KUKA KRL program: chk_w2_grp4_clo.src, chk_w2_grp4_clo.dat

--- chk_w2_grp4_clo.src ---
&ACCESS RV2
&REL 12
&COMMENT Check grampos Z4 fechado
&PARAM DISKPATH = Program/SubeRotine
&PARAM TEMPLATE = C:\KRC\Roboter\Template\vorgabe
&PARAM EDITMASK = *
DEF chk_w2_grp4_clo( )
;FOLD ; Programa de verificacao de grampos Z4 fechado;%{PE}%R 4.1.16,%MKUKATPBASIS,%CCOMMENT,%VNORMAL,%P 2:Programa de verificacao de grampos Z4 fechado
;ENDFOLD

$TIMER[10] = 0
$TIMER_STOP[10] = FALSE

;FOLD WAIT FOR ( NOT IN 497 'Pres pc 1 Axor_Atego/ ACTROS Z4.1 OPN' );%{PE}%R 8.2.24,%MKUKATPBASIS,%CEXT_WAIT_FOR,%VEXT_WAIT_FOR,%P 2:, 4:NOT, 5:$IN, 6:497, 7:Pres pc 1 Axor_Atego/ ACTROS Z4.1 OPN, 9:
WAIT FOR  (  NOT $IN[497] )
;ENDFOLD
;FOLD WAIT FOR ( NOT IN 511 'ACTROS Z4.2 OPN' );%{PE}%R 8.2.24,%MKUKATPBASIS,%CEXT_WAIT_FOR,%VEXT_WAIT_FOR,%P 2:, 4:NOT, 5:$IN, 6:511, 7:ACTROS Z4.2 OPN, 9:
WAIT FOR  (  NOT $IN[511] )
;ENDFOLD
;FOLD WAIT FOR ( NOT IN 517 'Z4.2 ABERTO/ ACTROS Z4.3 OPN' );%{PE}%R 8.2.24,%MKUKATPBASIS,%CEXT_WAIT_FOR,%VEXT_WAIT_FOR,%P 2:, 4:NOT, 5:$IN, 6:517, 7:Z4.2 ABERTO/ ACTROS Z4.3 OPN, 9:
WAIT FOR  (  NOT $IN[517] )
;ENDFOLD
;FOLD WAIT FOR ( NOT IN 519 'Z4.3 ABERTO/ ACTROS Z4.4 OPN' );%{PE}%R 8.2.24,%MKUKATPBASIS,%CEXT_WAIT_FOR,%VEXT_WAIT_FOR,%P 2:, 4:NOT, 5:$IN, 6:519, 7:Z4.3 ABERTO/ ACTROS Z4.4 OPN, 9:
WAIT FOR  (  NOT $IN[519] )
;ENDFOLD
;FOLD WAIT FOR ( IN 498 'Pres pc 2 Axor_Atego/ ACTROS Z4.1 CLO' );%{PE}%R 8.2.24,%MKUKATPBASIS,%CEXT_WAIT_FOR,%VEXT_WAIT_FOR,%P 2:, 4:, 5:$IN, 6:498, 7:Pres pc 2 Axor_Atego/ ACTROS Z4.1 CLO, 9:
WAIT FOR  ( $IN[498] )
;ENDFOLD
;FOLD WAIT FOR ( IN 512 'ACTROS Z4.2 CLO' );%{PE}%R 8.2.24,%MKUKATPBASIS,%CEXT_WAIT_FOR,%VEXT_WAIT_FOR,%P 2:, 4:, 5:$IN, 6:512, 7:ACTROS Z4.2 CLO, 9:
WAIT FOR  ( $IN[512] )
;ENDFOLD
;FOLD WAIT FOR ( IN 518 'Z4.2 FECHADO/ ACTROS Z4.3 CLO' );%{PE}%R 8.2.24,%MKUKATPBASIS,%CEXT_WAIT_FOR,%VEXT_WAIT_FOR,%P 2:, 4:, 5:$IN, 6:518, 7:Z4.2 FECHADO/ ACTROS Z4.3 CLO, 9:
WAIT FOR  ( $IN[518] )
;ENDFOLD
;FOLD WAIT FOR ( IN 520 'Z4.3 FECHADO/ ACTROS Z4.4 CLO' );%{PE}%R 8.2.24,%MKUKATPBASIS,%CEXT_WAIT_FOR,%VEXT_WAIT_FOR,%P 2:, 4:, 5:$IN, 6:520, 7:Z4.3 FECHADO/ ACTROS Z4.4 CLO, 9:
WAIT FOR  ( $IN[520] )
;ENDFOLD

$TIMER_STOP[10] = TRUE
$TIMER[10] = 0

END

--- chk_w2_grp4_clo.dat ---
&ACCESS RV2
&REL 12
&COMMENT Check grampos Z4 fechado
&PARAM DISKPATH = Program/SubeRotine
&PARAM TEMPLATE = C:\KRC\Roboter\Template\vorgabe
&PARAM EDITMASK = *
DEFDAT chk_w2_grp4_clo
;FOLD EXTERNAL DECLARATIONS;%{PE}%V3.2.0,%MKUKATPBASIS,%CEXT,%VCOMMON,%P
;FOLD BAS EXT;%{PE}%V3.2.0,%MKUKATPBASIS,%CEXT,%VEXT,%P
EXT  BAS (BAS_COMMAND  :IN,REAL  :IN )
DECL INT SUCCESS
;ENDFOLD
;FOLD GRIPPER EXT;%{E}%V3.2.0,%MKUKATPGRIPPER,%CEXT,%VEXT,%P
EXT  H50 (INT:IN, INT:IN ,INT:IN ,GRP_TYP:IN)
;ENDFOLD
;FOLD SPOT EXT;%{E}%V3.2.0,%MKUKATPSPOT,%CEXT,%VEXT,%P
EXT  USERSPOT (S_COMMAND  :IN, SPOT_TYPE:IN)
;ENDFOLD
;FOLD USER EXT;%{E}%V3.2.0,%MKUKATPUSER,%CEXT,%VEXT,%P
;Make here your modifications
;ENDFOLD
;ENDFOLD

ENDDAT
